TYPE "Positioning_MOL_Machine_Alr"
VERSION : 0.1
// Block: Positioning_MOL_Machine_Alr
   STRUCT
      Ax_NotHomed : Bool;
      Ax : OOAx_Alr;
      Motor : MotorSAlr;
   END_STRUCT;

END_TYPE
